FUNCTION_BLOCK TTestRunner 
VAR_INPUT
    RunTestsSequentially : BOOL;
END_VAR
VAR
    Run : BOOL := TRUE;
    
    State :(
        Init,
        RunTests_Concurrently,
        RunTests_Sequentially,
        CheckResults);
        
    i : INT;
    CompletedTestsCount : INT;
    FailedTestsCount : INT;
    CurrentTestIndex : INT;
    
    _TestsRunning : BOOL;
    _Results : T_MaxString;
    _AllTestsCompleted : BOOL;
    _TestCount : INT;
    
    Tests : ARRAY[0..MAX_TESTS] OF IUnitTest;
    TestResults : ARRAY[0..MAX_TESTS] OF TTestResult;
    AssertionMessages : TAssertionMessageList;
    
    TestsCompletedPercentage : LREAL;
END_VAR

CASE State OF
    Init:
        IF Run THEN
            Run := FALSE;
            ClearResults();
            AssertionMessages.Clear();
            FOR i := 0 TO _TestCount - 1 DO
                IF Tests[i] <> 0 THEN
                    Tests[i].Initialise(AssertionMessages);
				END_IF
			END_FOR
            _TestsRunning := TRUE;
            IF RunTestsSequentially THEN
                CurrentTestIndex := 0;
                State := RunTests_Sequentially;
            ELSE
                State := RunTests_Concurrently;
            END_IF
		END_IF
        
    RunTests_Concurrently:
        CompletedTestsCount := 0;
        FOR i := 0 TO _TestCount - 1 DO
            IF Tests[i] <> 0 THEN
                IF Tests[i].TestHasFinished THEN
                    addTimeStamp(TestResults[i]);
                    IF Tests[i].TestHasFailed THEN
                        TestResults[i].TestName  := Tests[i].TestName;
                        TestResults[i].TestState := 'Failed';
                        TestResults[i].ImageRef  := '3';
                        FailedTestsCount := FailedTestsCount + 1;
                    ELSE
                        TestResults[i].TestName  := Tests[i].TestName;
                        TestResults[i].TestState := 'Passed';
                        TestResults[i].ImageRef  := '2';
                    END_IF    
                    
                    CompletedTestsCount := CompletedTestsCount + 1;
                    TestsCompletedPercentage := CompletedTestsCount * 100/_TestCount;
                    _Results := F_FormatString2('%d Tests completed, %d Tests Failed',F_INT(CompletedTestsCount),F_INT(FailedTestsCount));
                ELSE
                    TestResults[i].TestName  := Tests[i].TestName;
                    TestResults[i].TestState := 'Running';
                    TestResults[i].ImageRef  := '1';
                    Tests[i].Execute();
                END_IF
            END_IF
        END_FOR
        IF CompletedTestsCount >= _TestCount THEN
            State := CheckResults;
		END_IF
        
    RunTests_Sequentially:
        IF Tests[CurrentTestIndex] <> 0 THEN
            IF Tests[CurrentTestIndex].TestHasFinished THEN
                addTimeStamp(TestResults[CurrentTestIndex]);
                IF Tests[CurrentTestIndex].TestHasFailed THEN
                    TestResults[CurrentTestIndex].TestName  := Tests[CurrentTestIndex].TestName;
                    TestResults[CurrentTestIndex].TestState := 'Failed';
                    TestResults[CurrentTestIndex].ImageRef  := '3';
                    FailedTestsCount := FailedTestsCount + 1;
                ELSE
                    TestResults[CurrentTestIndex].TestName  := Tests[CurrentTestIndex].TestName;
                    TestResults[CurrentTestIndex].TestState := 'Passed';
                    TestResults[CurrentTestIndex].ImageRef  := '2';
                END_IF    
                
                CompletedTestsCount := CompletedTestsCount + 1;
                CurrentTestIndex := CurrentTestIndex + 1;
                TestsCompletedPercentage := CompletedTestsCount * 100/_TestCount;
                _Results := F_FormatString2('%d Tests completed, %d Tests Failed',F_INT(CompletedTestsCount),F_INT(FailedTestsCount));
            ELSE
                TestResults[CurrentTestIndex].TestName  := Tests[CurrentTestIndex].TestName;
                TestResults[CurrentTestIndex].TestState := 'Running';
                TestResults[CurrentTestIndex].ImageRef  := '1';
                Tests[CurrentTestIndex].Execute();
            END_IF
        END_IF

        IF CompletedTestsCount >= _TestCount THEN
            State := CheckResults;
		END_IF

    CheckResults:
        _Results := F_FormatString2('%d Tests completed, %d Tests Failed',F_INT(CompletedTestsCount),F_INT(FailedTestsCount));
        _TestsRunning := FALSE;
        _AllTestsCompleted := TRUE;
        
        State := Init;
    
    
END_CASE

METHOD AddTest : BOOL
VAR_INPUT
    UnitTest : IUnitTest;
END_VAR
IF _TestCount < MAX_TESTS THEN
    Tests[_TestCount] := UnitTest;
    _TestCount := _TestCount + 1;
    AddTest := TRUE;
ELSE
    AssertionMessages.AddMessage('Maximum unit tests exceeded!');
END_IF
END_METHOD

METHOD PRIVATE addTimeStamp
VAR_IN_OUT
    TestResult : TTestResult;
END_VAR
VAR
	CurrentDcTime : T_DCTIME64;
    Now : TIMESTRUCT;
END_VAR
CurrentDcTime := F_GetActualDcTime64();
Now := DCTIME64_TO_SYSTEMTIME(CurrentDcTime);
TestResult.TestCompleteTime := tcl_StringUtils.F_TimeAsString_ms(Now);
END_METHOD

PROPERTY AllTestsCompleted : BOOL
GET
AllTestsCompleted := _AllTestsCompleted;
END_GET
END_PROPERTY

METHOD ClearResults
VAR_INPUT
END_VAR
_Results := '';
_AllTestsCompleted := FALSE;
FailedTestsCount := 0;
CompletedTestsCount := 0;
TestsCompletedPercentage := 0;

MEMSET(
    destAddr := ADR(TestResults), 
    fillByte := 0, 
    n        := SIZEOF(TestResults));
END_METHOD

PROPERTY Results : T_MaxString
GET
Results := _Results;
END_GET
END_PROPERTY

PROPERTY TestCount : INT
GET
TestCount := _TestCount;
END_GET
END_PROPERTY

PROPERTY TestsRunning : BOOL
GET
TestsRunning := _TestsRunning;
END_GET
END_PROPERTY

END_FUNCTION_BLOCK

(* stored: Version 1.1.0.1, ProductVersion 3.1.4024.4
   POU TTestRunner: Id {c7f35beb-7079-466d-ae1a-1beb011dea9f}, SpecialFunc None
   Method AddTest: Id {aff2d568-ab55-47bc-af2b-94e85ba5e218}
   Method addTimeStamp: Id {bdd169f4-a7c0-4197-b9c5-ebb28699c68a}
   Property AllTestsCompleted: Id {35232731-1165-473b-9489-dda727905bbe}
   Get Get: Id {427b4cbb-213d-4f37-80e2-9b36fbd84c82}
   Method ClearResults: Id {57179eef-fc7b-4bd0-85fd-730ca5472c60}
   Property Results: Id {d09ac635-f5a8-46e9-8513-febf5f67e4bf}
   Get Get: Id {bac56fdf-ab86-41b2-bda2-a53cd7cf550f}
   Property TestCount: Id {071111e2-ed4d-4d68-b95e-6b4cb6b3aa16}
   Get Get: Id {cc7bd08b-b6fe-4e09-88cb-16b9dd473b3f}
   Property TestsRunning: Id {cc8e65a0-6524-4f90-8531-cec392ab281c}
   Get Get: Id {0fb901a8-23b3-444c-a819-bc19c7f6c2c0} *)
